TYPE Control :
STRUCT
	Execute: BOOL;
	Send: BOOL;
	Update: BOOL;
	PixelCommand: Command;
END_STRUCT
END_TYPE

(* stored: Version 1.1.0.1, ProductVersion 3.1.4024.13
   DUT Control: Id {2044032a-37cc-4e9a-a599-15d7f6285cba} *)
